{attribute 'qualified_only'}
{attribute 'strict'}
TYPE VacuumGripper :
(
	on := 0,
	off
);
END_TYPE

(* stored: Version 1.1.0.1, ProductVersion 3.1.4022.12
   DUT VacuumGripper: Id {782a28a0-3dfe-4a5b-8079-62d2b95f0386} *)
